FUNCTION derivcvar_M_example_controller_t : LREAL
VAR_INPUT
	state: STATE;
END_VAR

derivcvar_M_example_controller_t := ifExprFunc1(state);

END_FUNCTION

(* stored: Version 1.1.0.1, ProductVersion 3.1.4022.18
   POU derivcvar_M_example_controller_t: Id {6a55c357-b588-4f9b-a165-6a252107f262}, SpecialFunc None *)
